FUNCTION_BLOCK FB_SeperateFileAndPathName
VAR_INPUT
	sPathAndFileName	:STRING(255);	// String with path and file name
END_VAR
VAR_OUTPUT
	sFileName			:STRING(80);	// String with file name
	sPathName			:STRING(175);	// String with path name
	bError				:BOOL;			// True if error occured during determination of file and path name
END_VAR
VAR
	iLength				:INT;			// Length of string that is examined
	iPos				:INT;			// Charactor position used to seperate file name from string
	iSize				:INT;			// Size of a string
	sTemp				:STRING;		// Temporary string
	iForIndex			:INT;			// Index used in for-loops
	bSeperatorFound		:BOOL;			// True if charator for folder seperator was found in input string
END_VAR


// Initialize flag for seperator found
bSeperatorFound := FALSE;

// Search through string and find the last "\" charactor
iLength := LEN(sPathAndFileName);
FOR iForIndex := 1 TO iLength BY 1 DO
	IF MID(sPathAndFileName,1,iForIndex) = '\' THEN
		iPos := iForIndex;
		bSeperatorFound := TRUE;
	END_IF
END_FOR

IF bSeperatorFound THEN
	// Set file name
	iSize := iLength - iPos;
	sFileName := RIGHT(sPathAndFileName,iSize);
	
	// Set path name
	sPathName := LEFT(sPathAndFileName,iPos);
	
	// Reset error flag
	bError := FALSE;
ELSE
	// Set error flag
	bError := TRUE;
END_IF

END_FUNCTION_BLOCK

(* stored: Version 1.1.0.1, ProductVersion 3.1.4024.12
   POU FB_SeperateFileAndPathName: Id {3bb7c6be-00c4-4233-b6b0-8ab3a16908cb}, SpecialFunc None *)
